// TIA Portal V16 export
// export: Created 2022-02-04T14:40:28.4340962Z, ExportSetting WithDefaults, DisplayName Totally Integrated Automation Portal, DisplayVersion V16 Update 1, DisplayName TIA Portal Version Control Interface, DisplayVersion V16, DisplayName TIA Portal Openness, DisplayVersion V16, DisplayName SINAMICS Startdrive Advanced, DisplayVersion V16 Update 5, DisplayName SINAMICS Startdrive G130, G150, S120, S150, SINAMICS MV, S210, DisplayVersion V16 Update 5, DisplayName SINAMICS Startdrive G110M, G120, G120C, G120D, G120P, G115D, DisplayVersion V16 Update 5, DisplayName STEP 7 Professional, DisplayVersion V16, DisplayName STEP 7 Safety, DisplayVersion V16, DisplayName WinCC Advanced, DisplayVersion V16, DisplayName SIMATIC Visualization Architect, DisplayVersion V16
TYPE "ServIM"
// stored: IsFailsafeCompliant false
   STRUCT
      BtnDU : Bool;   // Включить дистанционный режим
      BtnAU : Bool;   // Отключить дистанционный режим
      BtnFwd : Bool;   // Включить вперёд / выдвинуть
      BtnBwd : Bool;   // Включить назад / задвинуть
      BtnCmdStop : Bool;   // Остановить
      SetSpeedDU : Real;   // Задание на частотник в ДУ
      PrmBtnDU_ON : Bool;   // Разрешение на включение дистанционного режима
      PrmBtnDU_OF : Bool;   // Разрешение на отключение дистанционного режима
      PRMbtn_Back_ON : Bool;   // Разрешение кнопки включения заднего хода
      PRMbtn_Back_OFF : Bool;   // Разрешение кнопки отключения заднего хода
      PrmBtnCmdStop : Bool;   // Разрешение на остановку
      Ready : Bool;   // Готовность к работе
      ON : Bool;   // В работе
      OFF : Bool;   // Не в работе (закрыто)
      Fault : Bool;   // Обобщенная неисправность
      Alarm : Bool;   // Авария
      AU : Bool;   // Автоматическое управление
      MU : Bool;   // Местное управление
      DU : Bool;   // Дистанционный режим включен
      CMD_ON : Bool;   // Запустить ON
      CMD_OFF : Bool;   // Запустить OFF
      BACK : Bool;   // Реверс (задний ход)
      SetSpeed : Real;   // Задание на частотник
   END_STRUCT;
END_TYPE
